PROGRAM P_PersistentData
VAR
	writepersistent							: WRITEPERSISTENTDATA;
	bWrite									: BOOL;
	udiErrID								: UDINT;
END_VAR
VAR PERSISTENT
	iInt1									: INT:=10;
END_VAR

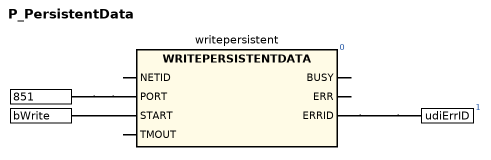
writepersistent(PORT := 851, START := bWrite); // WRITEPERSISTENTDATA
udiErrID := writepersistent.ERRID;

END_PROGRAM

(* stored: Version 1.1.0.1, ProductVersion 3.1.4022.7
   POU P_PersistentData: Id {5d2b5b0d-8c76-4509-bcc4-b9c1fe2cfb59}, SpecialFunc None *)
